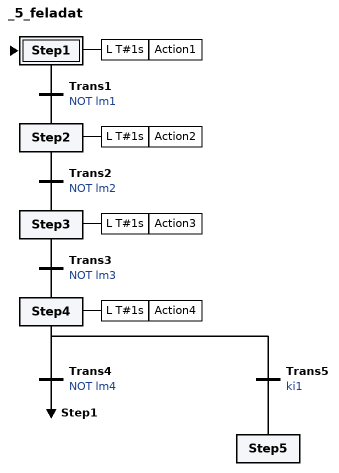
(* [picture p24: _5_feladat, sequence chart] *)
INITIAL_STEP Step1 :
Action1(L,T#1s) ;
END_STEP
TRANSITION Trans1 FROM Step1 TO Step2
 := NOT lm1;
END_TRANSITION
STEP Step2 :
Action2(L,T#1s) ;
END_STEP
TRANSITION Trans2 FROM Step2 TO Step3
 := NOT lm2;
END_TRANSITION
STEP Step3 :
Action3(L,T#1s) ;
END_STEP
TRANSITION Trans3 FROM Step3 TO Step4
 := NOT lm3;
END_TRANSITION
STEP Step4 :
Action4(L,T#1s) ;
END_STEP
TRANSITION Trans4 (PRIORITY := 1) FROM Step4 TO Step1
 := NOT lm4;
END_TRANSITION
TRANSITION Trans5 (PRIORITY := 2) FROM Step4 TO Step5
 := ki1;
END_TRANSITION
STEP Step5 :
END_STEP

### Action Action4

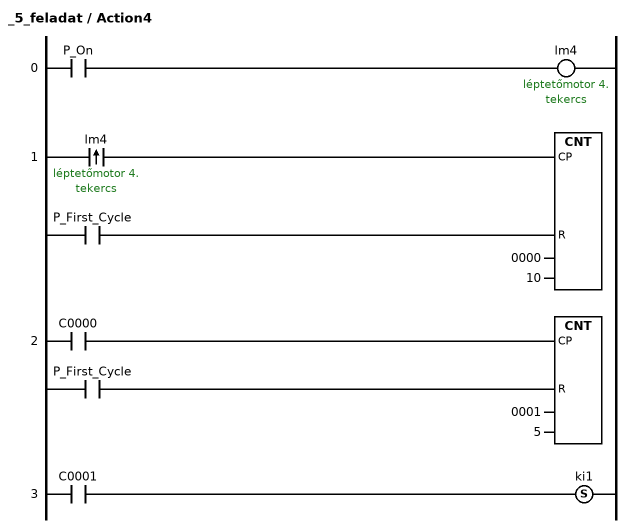
; rung 0
LD P_On
OUT lm4  ; léptetőmotor 4. tekercs
; rung 1
@LD lm4  ; léptetőmotor 4. tekercs
LD P_First_Cycle
CNT 0000 10
; rung 2
LD C0000
LD P_First_Cycle
CNT 0001 5
; rung 3
LD C0001
SET ki1

### Action Action3

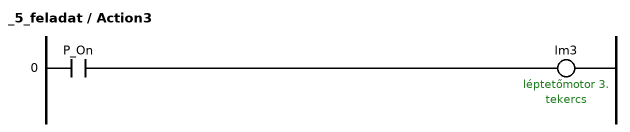
; rung 0
LD P_On
OUT lm3  ; léptetőmotor 3. tekercs

### Action Action2

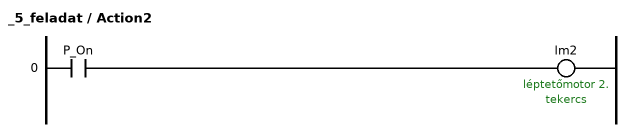
; rung 0
LD P_On
OUT lm2  ; léptetőmotor 2. tekercs

### Action Action1

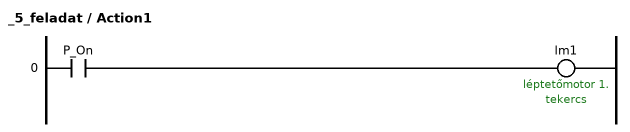
; rung 0
LD P_On
OUT lm1  ; léptetőmotor 1. tekercs

## Program _szorgalmi1 (interrupt task -1)
Local symbols
be1 0.00 BOOL
be2 0.01 BOOL
lm1 1.01 BOOL  ; léptetőmotor 1. tekercs
lm2 1.03 BOOL  ; léptetőmotor 2. tekercs
lm3 1.05 BOOL  ; léptetőmotor 3. tekercs
lm4 1.07 BOOL  ; léptetőmotor 4. tekercs
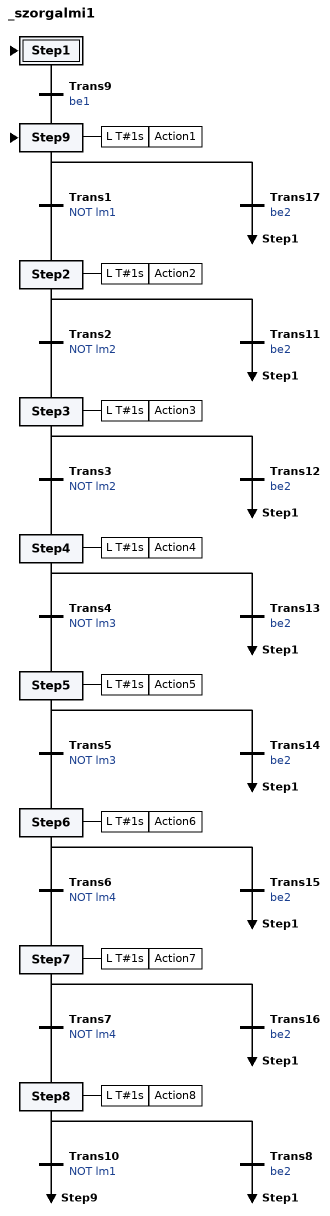
INITIAL_STEP Step1 :
END_STEP
STEP Step2 :
Action2(L,T#1s) ;
END_STEP
STEP Step3 :
Action3(L,T#1s) ;
END_STEP
STEP Step4 :
Action4(L,T#1s) ;
END_STEP
STEP Step5 :
Action5(L,T#1s) ;
END_STEP
STEP Step6 :
Action6(L,T#1s) ;
END_STEP
STEP Step7 :
Action7(L,T#1s) ;
END_STEP
STEP Step8 :
Action8(L,T#1s) ;
END_STEP
TRANSITION Trans9 FROM Step1 TO Step9
 := be1;
END_TRANSITION
STEP Step9 :
Action1(L,T#1s) ;
END_STEP
TRANSITION Trans10 (PRIORITY := 1) FROM Step8 TO Step9
 := NOT lm1;
END_TRANSITION
TRANSITION Trans8 (PRIORITY := 2) FROM Step8 TO Step1
 := be2;
END_TRANSITION
TRANSITION Trans2 (PRIORITY := 1) FROM Step2 TO Step3
 := NOT lm2;
END_TRANSITION
TRANSITION Trans11 (PRIORITY := 2) FROM Step2 TO Step1
 := be2;
END_TRANSITION
TRANSITION Trans3 (PRIORITY := 1) FROM Step3 TO Step4
 := NOT lm2;
END_TRANSITION
TRANSITION Trans12 (PRIORITY := 2) FROM Step3 TO Step1
 := be2;
END_TRANSITION
TRANSITION Trans4 (PRIORITY := 1) FROM Step4 TO Step5
 := NOT lm3;
END_TRANSITION
TRANSITION Trans13 (PRIORITY := 2) FROM Step4 TO Step1
 := be2;
END_TRANSITION
TRANSITION Trans5 (PRIORITY := 1) FROM Step5 TO Step6
 := NOT lm3;
END_TRANSITION
TRANSITION Trans14 (PRIORITY := 2) FROM Step5 TO Step1
 := be2;
END_TRANSITION
TRANSITION Trans6 (PRIORITY := 1) FROM Step6 TO Step7
 := NOT lm4;
END_TRANSITION
TRANSITION Trans15 (PRIORITY := 2) FROM Step6 TO Step1
 := be2;
END_TRANSITION
TRANSITION Trans7 (PRIORITY := 1) FROM Step7 TO Step8
 := NOT lm4;
END_TRANSITION
TRANSITION Trans16 (PRIORITY := 2) FROM Step7 TO Step1
 := be2;
END_TRANSITION
TRANSITION Trans1 (PRIORITY := 1) FROM Step9 TO Step2
 := NOT lm1;
END_TRANSITION
TRANSITION Trans17 (PRIORITY := 2) FROM Step9 TO Step1
 := be2;
END_TRANSITION

### Action Action8

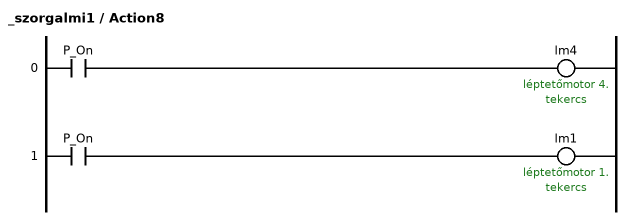
; rung 0
LD P_On
OUT lm4  ; léptetőmotor 4. tekercs
; rung 1
LD P_On
OUT lm1  ; léptetőmotor 1. tekercs

### Action Action7

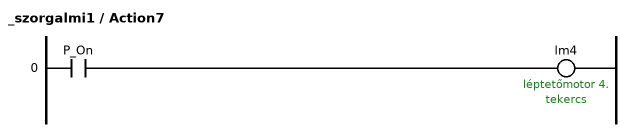
; rung 0
LD P_On
OUT lm4  ; léptetőmotor 4. tekercs

### Action Action6

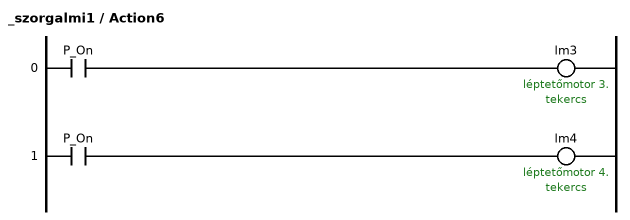
; rung 0
LD P_On
OUT lm3  ; léptetőmotor 3. tekercs
; rung 1
LD P_On
OUT lm4  ; léptetőmotor 4. tekercs

### Action Action5

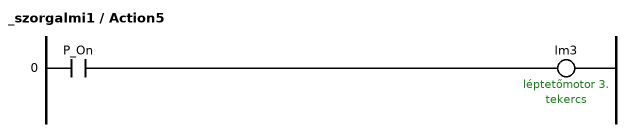
; rung 0
LD P_On
OUT lm3  ; léptetőmotor 3. tekercs

### Action Action4

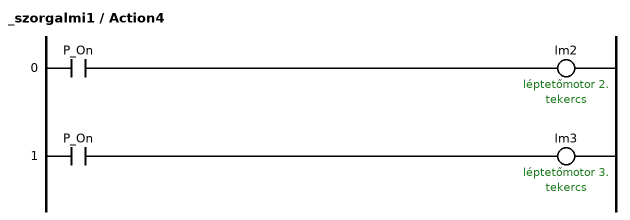
; rung 0
LD P_On
OUT lm2  ; léptetőmotor 2. tekercs
; rung 1
LD P_On
OUT lm3  ; léptetőmotor 3. tekercs

### Action Action3

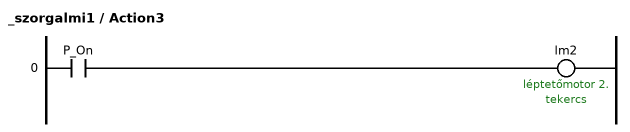
; rung 0
LD P_On
OUT lm2  ; léptetőmotor 2. tekercs

### Action Action2

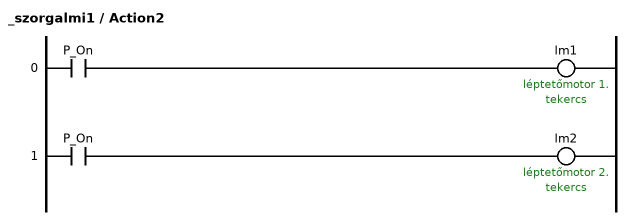
; rung 0
LD P_On
OUT lm1  ; léptetőmotor 1. tekercs
; rung 1
LD P_On
OUT lm2  ; léptetőmotor 2. tekercs

### Action Action1

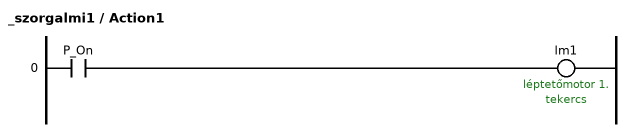
; rung 0
LD P_On
OUT lm1  ; léptetőmotor 1. tekercs

### Action Action9

## Program _szorgalmi2 (interrupt task -1)
Local symbols
be5 0.04 BOOL
be6 0.05 BOOL
lm1 1.01 BOOL  ; léptetőmotor 1. tekercs
lm2 1.03 BOOL  ; léptetőmotor 2. tekercs
lm3 1.05 BOOL  ; léptetőmotor 3. tekercs
lm4 1.07 BOOL  ; léptetőmotor 4. tekercs
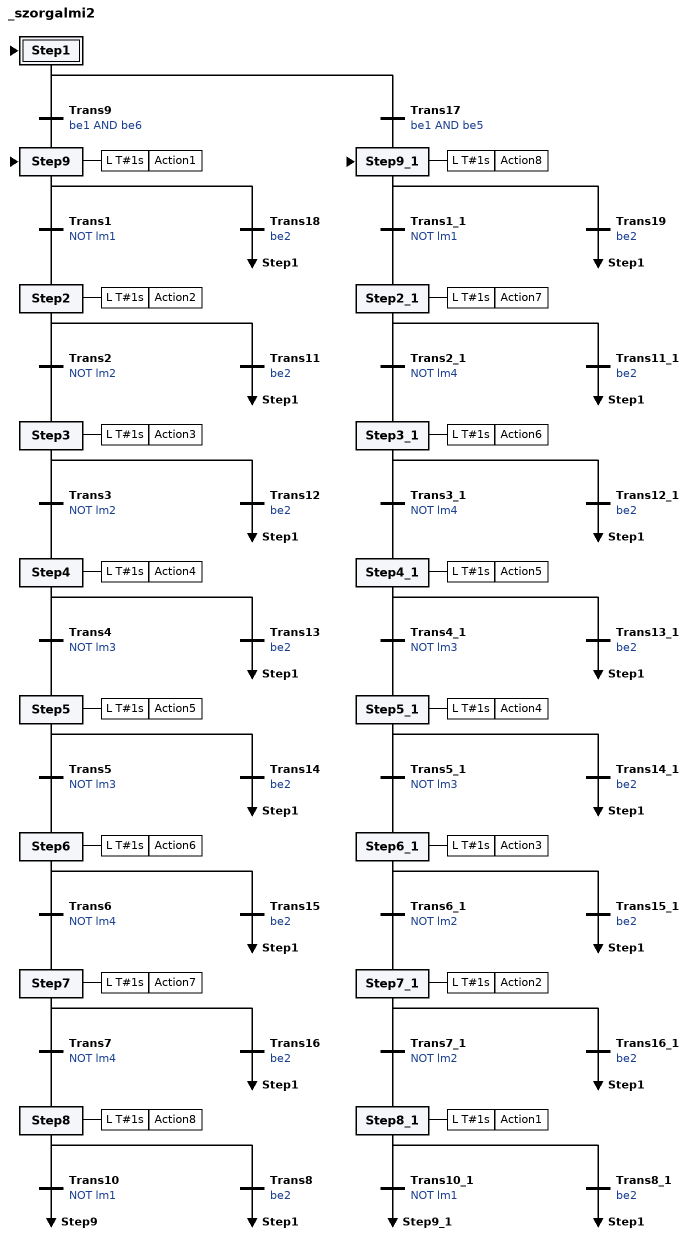
INITIAL_STEP Step1 :
END_STEP
STEP Step2 :
Action2(L,T#1s) ;
END_STEP
STEP Step3 :
Action3(L,T#1s) ;
END_STEP
STEP Step4 :
Action4(L,T#1s) ;
END_STEP
STEP Step5 :
Action5(L,T#1s) ;
END_STEP
STEP Step6 :
Action6(L,T#1s) ;
END_STEP
STEP Step7 :
Action7(L,T#1s) ;
END_STEP
STEP Step8 :
Action8(L,T#1s) ;
END_STEP
STEP Step9 :
Action1(L,T#1s) ;
END_STEP
TRANSITION Trans10 (PRIORITY := 1) FROM Step8 TO Step9
 := NOT lm1;
END_TRANSITION
TRANSITION Trans8 (PRIORITY := 2) FROM Step8 TO Step1
 := be2;
END_TRANSITION
TRANSITION Trans2 (PRIORITY := 1) FROM Step2 TO Step3
 := NOT lm2;
END_TRANSITION
TRANSITION Trans11 (PRIORITY := 2) FROM Step2 TO Step1
 := be2;
END_TRANSITION
TRANSITION Trans3 (PRIORITY := 1) FROM Step3 TO Step4
 := NOT lm2;
END_TRANSITION
TRANSITION Trans12 (PRIORITY := 2) FROM Step3 TO Step1
 := be2;
END_TRANSITION
TRANSITION Trans4 (PRIORITY := 1) FROM Step4 TO Step5
 := NOT lm3;
END_TRANSITION
TRANSITION Trans13 (PRIORITY := 2) FROM Step4 TO Step1
 := be2;
END_TRANSITION
TRANSITION Trans5 (PRIORITY := 1) FROM Step5 TO Step6
 := NOT lm3;
END_TRANSITION
TRANSITION Trans14 (PRIORITY := 2) FROM Step5 TO Step1
 := be2;
END_TRANSITION
TRANSITION Trans6 (PRIORITY := 1) FROM Step6 TO Step7
 := NOT lm4;
END_TRANSITION
TRANSITION Trans15 (PRIORITY := 2) FROM Step6 TO Step1
 := be2;
END_TRANSITION
TRANSITION Trans7 (PRIORITY := 1) FROM Step7 TO Step8
 := NOT lm4;
END_TRANSITION
TRANSITION Trans16 (PRIORITY := 2) FROM Step7 TO Step1
 := be2;
END_TRANSITION
TRANSITION Trans9 (PRIORITY := 1) FROM Step1 TO Step9
 := be1 AND be6;
END_TRANSITION
TRANSITION Trans17 (PRIORITY := 2) FROM Step1 TO Step9_1
 := be1 AND be5;
END_TRANSITION
STEP Step2_1 :
Action7(L,T#1s) ;
END_STEP
STEP Step3_1 :
Action6(L,T#1s) ;
END_STEP
STEP Step4_1 :
Action5(L,T#1s) ;
END_STEP
STEP Step5_1 :
Action4(L,T#1s) ;
END_STEP
STEP Step6_1 :
Action3(L,T#1s) ;
END_STEP
STEP Step7_1 :
Action2(L,T#1s) ;
END_STEP
STEP Step8_1 :
Action1(L,T#1s) ;
END_STEP
STEP Step9_1 :
Action8(L,T#1s) ;
END_STEP
TRANSITION Trans10_1 (PRIORITY := 1) FROM Step8_1 TO Step9_1
 := NOT lm1;
END_TRANSITION
TRANSITION Trans8_1 (PRIORITY := 2) FROM Step8_1 TO Step1
 := be2;
END_TRANSITION
TRANSITION Trans2_1 (PRIORITY := 1) FROM Step2_1 TO Step3_1
 := NOT lm4;
END_TRANSITION
TRANSITION Trans11_1 (PRIORITY := 2) FROM Step2_1 TO Step1
 := be2;
END_TRANSITION
TRANSITION Trans3_1 (PRIORITY := 1) FROM Step3_1 TO Step4_1
 := NOT lm4;
END_TRANSITION
TRANSITION Trans12_1 (PRIORITY := 2) FROM Step3_1 TO Step1
 := be2;
END_TRANSITION
TRANSITION Trans4_1 (PRIORITY := 1) FROM Step4_1 TO Step5_1
 := NOT lm3;
END_TRANSITION
TRANSITION Trans13_1 (PRIORITY := 2) FROM Step4_1 TO Step1
 := be2;
END_TRANSITION
TRANSITION Trans5_1 (PRIORITY := 1) FROM Step5_1 TO Step6_1
 := NOT lm3;
END_TRANSITION
TRANSITION Trans14_1 (PRIORITY := 2) FROM Step5_1 TO Step1
 := be2;
END_TRANSITION
TRANSITION Trans6_1 (PRIORITY := 1) FROM Step6_1 TO Step7_1
 := NOT lm2;
END_TRANSITION
TRANSITION Trans15_1 (PRIORITY := 2) FROM Step6_1 TO Step1
 := be2;
END_TRANSITION
TRANSITION Trans7_1 (PRIORITY := 1) FROM Step7_1 TO Step8_1
 := NOT lm2;
END_TRANSITION
TRANSITION Trans16_1 (PRIORITY := 2) FROM Step7_1 TO Step1
 := be2;
END_TRANSITION
TRANSITION Trans1 (PRIORITY := 1) FROM Step9 TO Step2
 := NOT lm1;
END_TRANSITION
TRANSITION Trans18 (PRIORITY := 2) FROM Step9 TO Step1
 := be2;
END_TRANSITION
TRANSITION Trans1_1 (PRIORITY := 1) FROM Step9_1 TO Step2_1
 := NOT lm1;
END_TRANSITION
TRANSITION Trans19 (PRIORITY := 2) FROM Step9_1 TO Step1
 := be2;
END_TRANSITION

### Action Action1

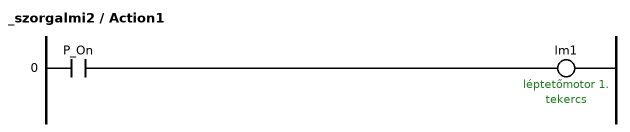
; rung 0
LD P_On
OUT lm1  ; léptetőmotor 1. tekercs

### Action Action2

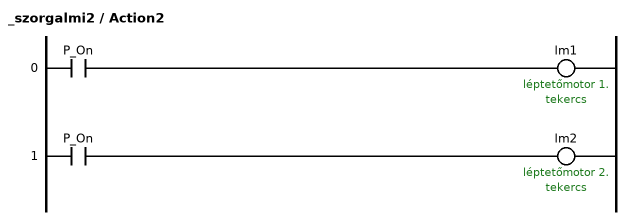
; rung 0
LD P_On
OUT lm1  ; léptetőmotor 1. tekercs
; rung 1
LD P_On
OUT lm2  ; léptetőmotor 2. tekercs

### Action Action3

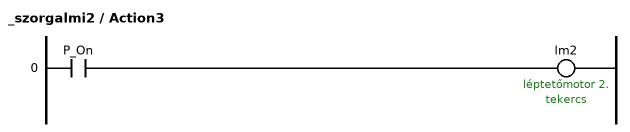
; rung 0
LD P_On
OUT lm2  ; léptetőmotor 2. tekercs

### Action Action4

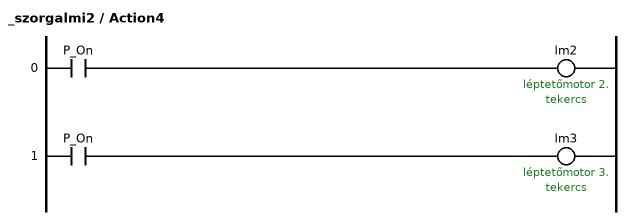
; rung 0
LD P_On
OUT lm2  ; léptetőmotor 2. tekercs
; rung 1
LD P_On
OUT lm3  ; léptetőmotor 3. tekercs

### Action Action5

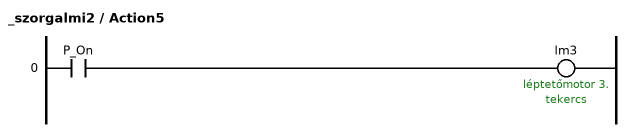
; rung 0
LD P_On
OUT lm3  ; léptetőmotor 3. tekercs

### Action Action6

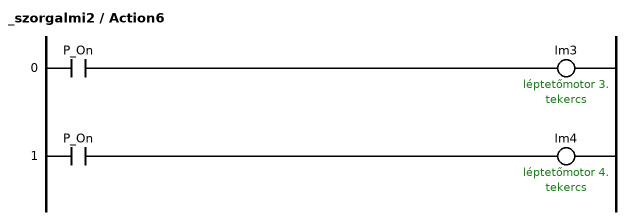
; rung 0
LD P_On
OUT lm3  ; léptetőmotor 3. tekercs
; rung 1
LD P_On
OUT lm4  ; léptetőmotor 4. tekercs

### Action Action7

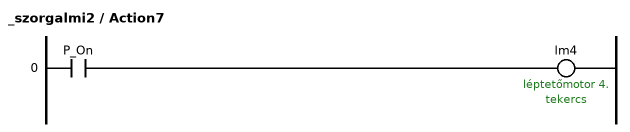
; rung 0
LD P_On
OUT lm4  ; léptetőmotor 4. tekercs

### Action Action8

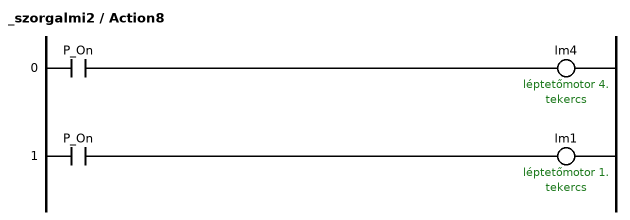
; rung 0
LD P_On
OUT lm4  ; léptetőmotor 4. tekercs
; rung 1
LD P_On
OUT lm1  ; léptetőmotor 1. tekercs

### Action Action9

### Action Action10